// TIA Portal V20 export
ORGANIZATION_BLOCK "Main"   // OB1, LAD, ProgramCycle
TITLE = "Main Program Sweep (Cycle)"
{ S7_Optimized_Access := 'TRUE' }
// stored: SetENOAutomatically false
   VAR_INPUT
      Initial_Call : Bool;   // Initial call of this OB
      Remanence : Bool;   // =True, if remanent data are available
   END_VAR
BEGIN

REGION Network 1
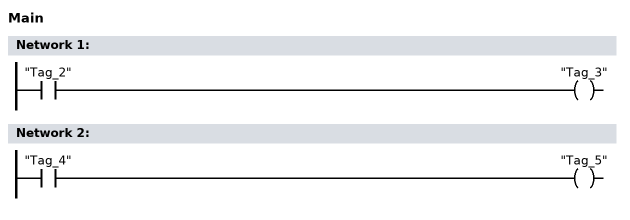
   RUNG wire#powerrail
      Contact( "Tag_2" )
      Coil( "Tag_3" )
   END_RUNG
   // the same network as SCL:
   "Tag_3" := "Tag_2";
END_REGION

REGION Network 2
   RUNG wire#powerrail
      Contact( "Tag_4" )
      Coil( "Tag_5" )
   END_RUNG
   // the same network as SCL:
   "Tag_5" := "Tag_4";
END_REGION
END_ORGANIZATION_BLOCK
